// Type alias for a single character string.
TYPE T_Char : STRING(1); END_TYPE

(* stored: Version 1.1.0.1
   DUT T_Char: Id {3574fb77-fae6-08e6-181c-545816d08d50} *)
